% RSLogix 500 project P3_IVANOVSKI_M.RSS, saved by version 8.30.00.16 %
PROJECT "UNTITLED"    % processor: Bul.1763 MicroLogix 1100 Series B %

PROGRAM FILES
  LAD 2 "MAIN"  5 rungs
  LAD 3 "BARCD INFO"  4 rungs
  LAD 4 "COMPUTE"  9 rungs

DATA FILES
  O0 OUTPUT  4 elements
  I1 INPUT  6 elements
  S2 STATUS  66 elements
  B3 BINARY  1 elements
  T4 TIMER  1 elements
  C5 COUNTER  1 elements
  R6 CONTROL  1 elements
  N7 INTEGER  15 elements
  F8 FLOAT  1 elements
  ST9 STRING  10 elements  % BARCODE SCAN %

LADDER 2 "MAIN"
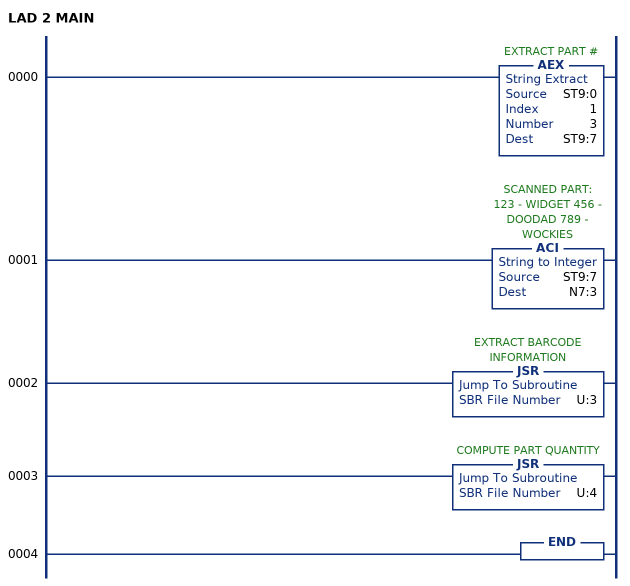
% Rung: 0 %
SOR AEX ST9:0 1 3 ST9:7 EOR
%   ST9:0  "PPP-QQ-D" %
%   ST9:7  "EXTRACT PART #" %
% Rung: 1 %
SOR ACI ST9:7 N7:3 EOR
%   ST9:7  "EXTRACT PART #" %
%   N7:3  "SCANNED PART: 123 - WIDGET 456 - DOODAD 789 - WOCKIES" %
% Rung: 2 %
SOR JSR U:3 EOR
%   U:3  "EXTRACT BARCODE INFORMATION" %
% Rung: 3 %
SOR JSR U:4 EOR
%   U:4  "COMPUTE PART QUANTITY" %
% Rung: 4 %
SOR END EOR

LADDER 3 "BARCD INFO"
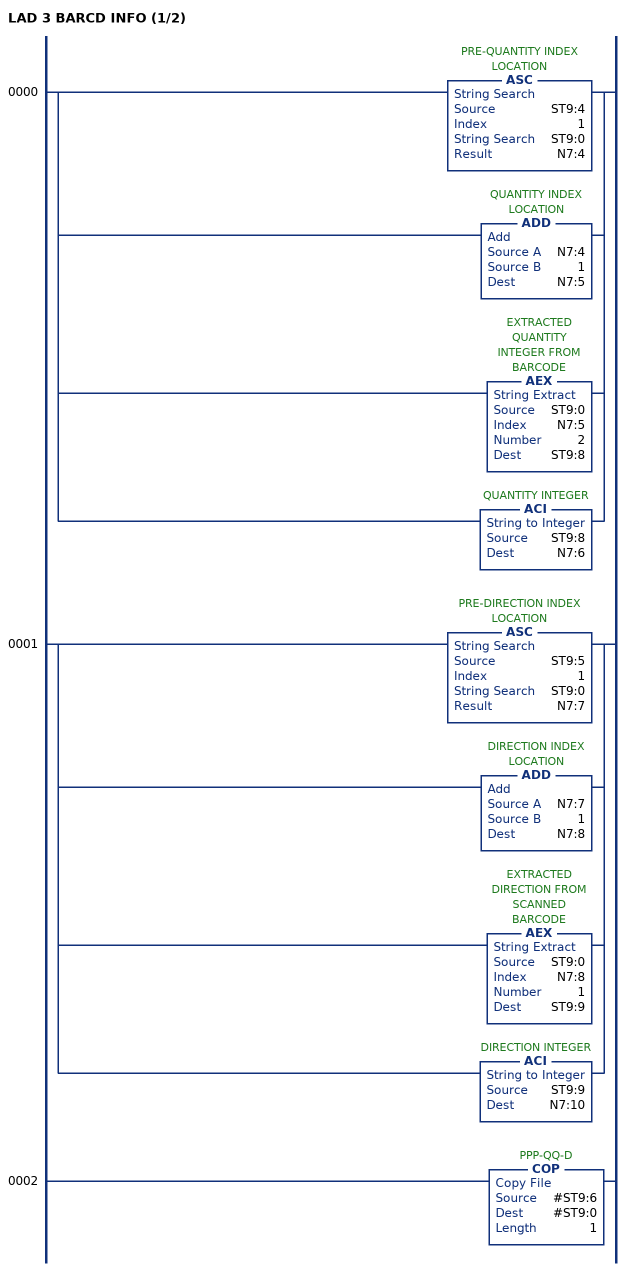
% Rung: 0 %
SOR BST ASC ST9:4 1 ST9:0 N7:4 NXB ADD N7:4 1 N7:5 NXB AEX ST9:0 N7:5 2 ST9:8 NXB ACI ST9:8 N7:6 BND EOR
%   ST9:4  "PRE-QUANTITY INDEX LOCATION" %
%   ST9:0  "PPP-QQ-D" %
%   N7:4  "PRE-QUANTITY INDEX LOCATION" %
%   N7:5  "QUANTITY INDEX LOCATION" %
%   ST9:8  "EXTRACTED QUANTITY INTEGER FROM BARCODE" %
%   N7:6  "QUANTITY INTEGER" %
% Rung: 1 %
SOR BST ASC ST9:5 1 ST9:0 N7:7 NXB ADD N7:7 1 N7:8 NXB AEX ST9:0 N7:8 1 ST9:9 NXB ACI ST9:9 N7:10 BND EOR
%   ST9:5  "PRE-DIRECTION INDEX LOCATION" %
%   ST9:0  "PPP-QQ-D" %
%   N7:7  "PRE-DIRECTION INDEX LOCATION" %
%   N7:8  "DIRECTION INDEX LOCATION" %
%   ST9:9  "EXTRACTED DIRECTION FROM SCANNED BARCODE" %
%   N7:10  "DIRECTION INTEGER" %
% Rung: 2 %
SOR COP #ST9:6 #ST9:0 1 EOR
%   ST9:6  "CLEAR SCANNED BARCODE" %
%   ST9:0  "PPP-QQ-D" %

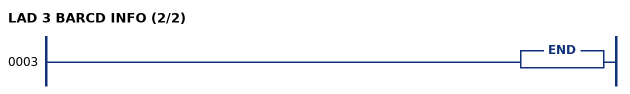
% Rung: 3 %
SOR END EOR

LADDER 4 "COMPUTE"
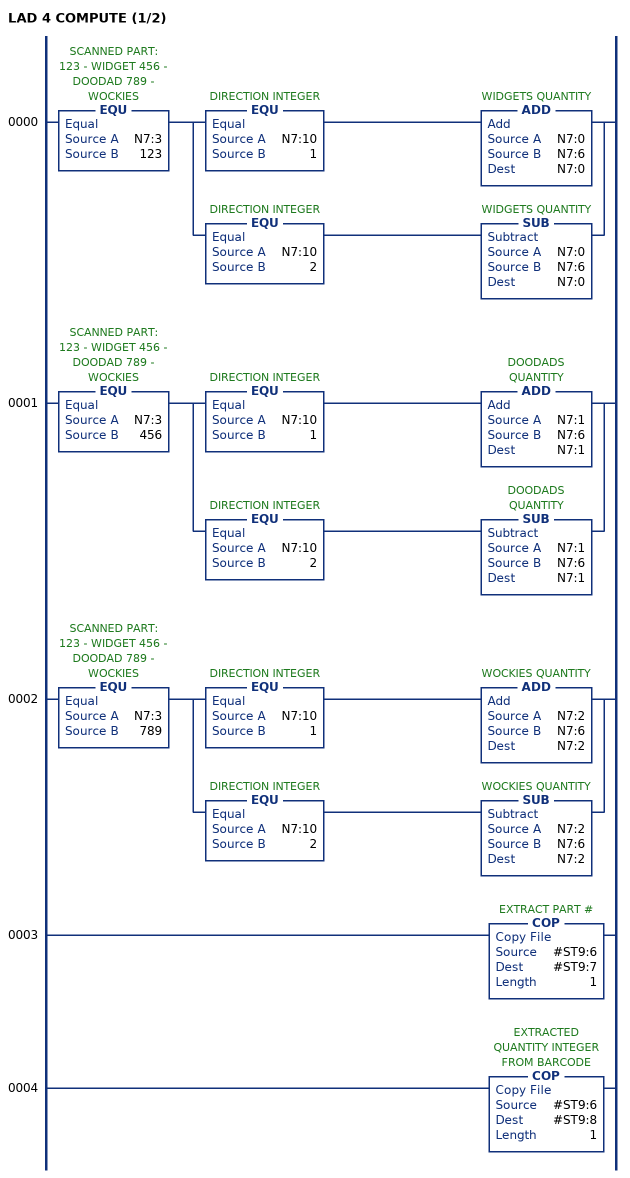
% Rung: 0 %
SOR EQU N7:3 123 BST EQU N7:10 1 ADD N7:0 N7:6 N7:0 NXB EQU N7:10 2 SUB N7:0 N7:6 N7:0 BND EOR
%   N7:3  "SCANNED PART: 123 - WIDGET 456 - DOODAD 789 - WOCKIES" %
%   N7:10  "DIRECTION INTEGER" %
%   N7:0  "WIDGETS QUANTITY" %
%   N7:6  "QUANTITY INTEGER" %
% Rung: 1 %
SOR EQU N7:3 456 BST EQU N7:10 1 ADD N7:1 N7:6 N7:1 NXB EQU N7:10 2 SUB N7:1 N7:6 N7:1 BND EOR
%   N7:3  "SCANNED PART: 123 - WIDGET 456 - DOODAD 789 - WOCKIES" %
%   N7:10  "DIRECTION INTEGER" %
%   N7:1  "DOODADS QUANTITY" %
%   N7:6  "QUANTITY INTEGER" %
% Rung: 2 %
SOR EQU N7:3 789 BST EQU N7:10 1 ADD N7:2 N7:6 N7:2 NXB EQU N7:10 2 SUB N7:2 N7:6 N7:2 BND EOR
%   N7:3  "SCANNED PART: 123 - WIDGET 456 - DOODAD 789 - WOCKIES" %
%   N7:10  "DIRECTION INTEGER" %
%   N7:2  "WOCKIES QUANTITY" %
%   N7:6  "QUANTITY INTEGER" %
% Rung: 3 %
SOR COP #ST9:6 #ST9:7 1 EOR
%   ST9:6  "CLEAR SCANNED BARCODE" %
%   ST9:7  "EXTRACT PART #" %
% Rung: 4 %
SOR COP #ST9:6 #ST9:8 1 EOR
%   ST9:6  "CLEAR SCANNED BARCODE" %
%   ST9:8  "EXTRACTED QUANTITY INTEGER FROM BARCODE" %

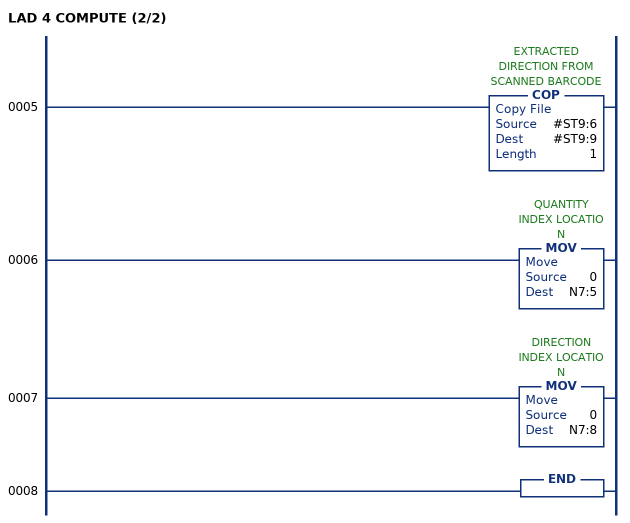
% Rung: 5 %
SOR COP #ST9:6 #ST9:9 1 EOR
%   ST9:6  "CLEAR SCANNED BARCODE" %
%   ST9:9  "EXTRACTED DIRECTION FROM SCANNED BARCODE" %
% Rung: 6 %
SOR MOV 0 N7:5 EOR
%   N7:5  "QUANTITY INDEX LOCATION" %
% Rung: 7 %
SOR MOV 0 N7:8 EOR
%   N7:8  "DIRECTION INDEX LOCATION" %
% Rung: 8 %
SOR END EOR

OTHER DOCUMENTED ADDRESSES
  B3:0/0  "ONS"
  B3:0/1  "ONS"
  B3:0/2  "ONS"
  B3:0/3  "ONS"
  B3:0/4  "ONS"
  B3:0/5  "ONS"
  B3:0/6  "ONS"
  B3:0/7  "ONS"
  B3:0/8  "ONS"
  N7:3/0  "CLEAR PART NUMBER"
  N7:9  "DIRECTION INTEGER"
  N7:13  "DIRECTION: 1 - INCOMING 2 - OUTGOING"
  Q0:0  "WIDGET QTY COMPUTATION"
  Q2:1  "CLEAR STRING IF INCORRECT PART NUMBER"
  Q3:0  "WIDGET QTY COMPUTATION"
  Q3:1  Q3
  Q4:0  "WIDGET QTY COMPUTATION"
  ST9:1  "WIDGET PART NUMBER"
  ST9:2  "DOODADS PART NUMBER"
  ST9:3  "WOCKIES PART NUMBER"
  WIDGET  "WIDGET QTY COMPUTATION"

DATA TABLE (non-zero values as saved)
DATA B3
% B3:0 % 0X003F
DATA ST9
% ST9:1 % "123"
% ST9:2 % "456"
% ST9:3 % "789"
% ST9:4 % "-"
% ST9:5 % ":"
